FUNCTION_BLOCK FB_Emg_Stop
VAR_INPUT
END_VAR
VAR_OUTPUT
END_VAR
VAR
END_VAR

END_FUNCTION_BLOCK

(* stored: Version 1.1.0.1, ProductVersion 3.1.4024.13
   POU FB_Emg_Stop: Id {6cda912b-c67a-4d63-a638-3cc993734bb7}, SpecialFunc None *)
